PROGRAM EM02_Placing1
VAR
	
	//Backbone
	FB_StateMachine_Placing1		: FB_StateManager;
	bFl_RunningMachinePlacing1		: BOOL;
	bFl_SeqReset					: BOOL;
	bFl_Manual						: BOOL;
	CheckStatusPlacing1				: checkstatus;
	AlarmEventHistory				: ARRAY[1..20] OF Alarm_Event_History;
	Placing1_Management				: FB_Placing_v2;
	bFl_Flushing					: BOOL;
	PalletID_Placing1				: PalletID_name;
	Placing1_ID						: STRING;
	bFl_PalletJammed				: BOOL;
	
	//Motor
	Motor_PalletPlacing1			: MotorManagement;
	bFl_MotorPlacing1				: BOOL;
	Motor_Placing1_Error			: BOOL;
	Motor_Placing1_ErrorID			: UINT;
	bFl_MotorPlacing1_Fwd			: BOOL;
	bFl_MotorPlacing1_Rev			: BOOL;
	bFL_Safety						: BOOL;
	AlarmEventActive				: ARRAY[1..20] OF Alarm_Event_Active;
	CheckAcc						: TON;
END_VAR
VAR // added by the converter: edge detectors and wires of the graphical bodies
    _w1 : BOOL;
END_VAR

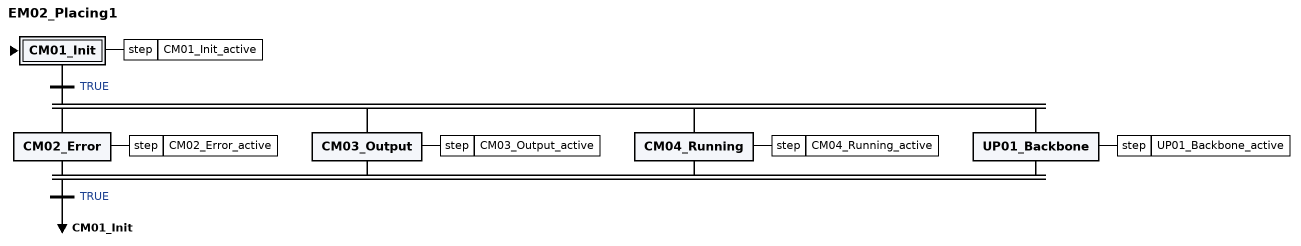
INITIAL_STEP CM01_Init:
    CM01_Init_active(N);  // step action
END_STEP
TRANSITION FROM CM01_Init TO (CM02_Error, CM03_Output, CM04_Running, UP01_Backbone)
    := TRUE;
END_TRANSITION
STEP CM02_Error:
    CM02_Error_active(N);  // step action
END_STEP
STEP CM03_Output:
    CM03_Output_active(N);  // step action
END_STEP
STEP CM04_Running:
    CM04_Running_active(N);  // step action
END_STEP
STEP UP01_Backbone:
    UP01_Backbone_active(N);  // step action
END_STEP
TRANSITION FROM (CM02_Error, CM03_Output, CM04_Running, UP01_Backbone) TO CM01_Init
    := TRUE;
END_TRANSITION

ACTION CM01_Init_active:
Data_GVL.bFL_StartPlacing1			:= Status_GVL.bFl_RunButton_Robotic OR HMI_GVL.bStartButtonPlacing1;
Data_GVL.bFL_StopPlacing1			:= NOT Status_GVL.bFl_StopButton_Robotic OR HMI_GVL.bStopButtonPlacing1;
Data_GVL.bFL_ResetPlacing1			:= Status_GVL.bFl_ResetButton_Robotic OR HMI_GVL.bResetButtonPlacing1;
Data_GVL.bFL_AckPlacing1			:= Status_GVL.bFl_Acknowledge_Robotic OR HMI_GVL.bAcknowledgeButtonPlacing1;
Data_GVL.bFL_AutoManuaModePlacing1 	:= Status_GVL.bFl_Manual_Robotic OR HMI_GVL.bTestModeEnablePlacing1;
bFl_RunningMachinePlacing1			:= Data_GVL.stStateMachinePlacing1.Running;
bFl_Manual							:= Data_GVL.stStateMachinePlacing1.ManualMode;
bFl_SeqReset						:= NOT Status_GVL.bFl_EStop_Robotic;
bFL_Safety							:= Status_GVL.bFl_EStop_Robotic AND Status_GVL.bSafety_DoorRobotic;


(*=================Convert Timer============================*)
Data_GVL.Tmr_Placing1	:= ConvertMilliSecTimeData(HMI_GVL.Tmr_Placing1);

(*=================Data OEE============================*)
Data_GVL.dt_Production[1].Data1			:= HMI_GVL.arCountTotal[1];
Data_GVL.dt_Production[1].Data2			:= HMI_GVL.arPalletTotal[1];
Data_GVL.dt_Production[1].Data3			:= HMI_GVL.arPalletIncomplete[1];
Data_GVL.dt_Production[1].ProductCode	:= Status_GVL.RecipeLine[1].ProductName;
END_ACTION

ACTION CM02_Error_active:
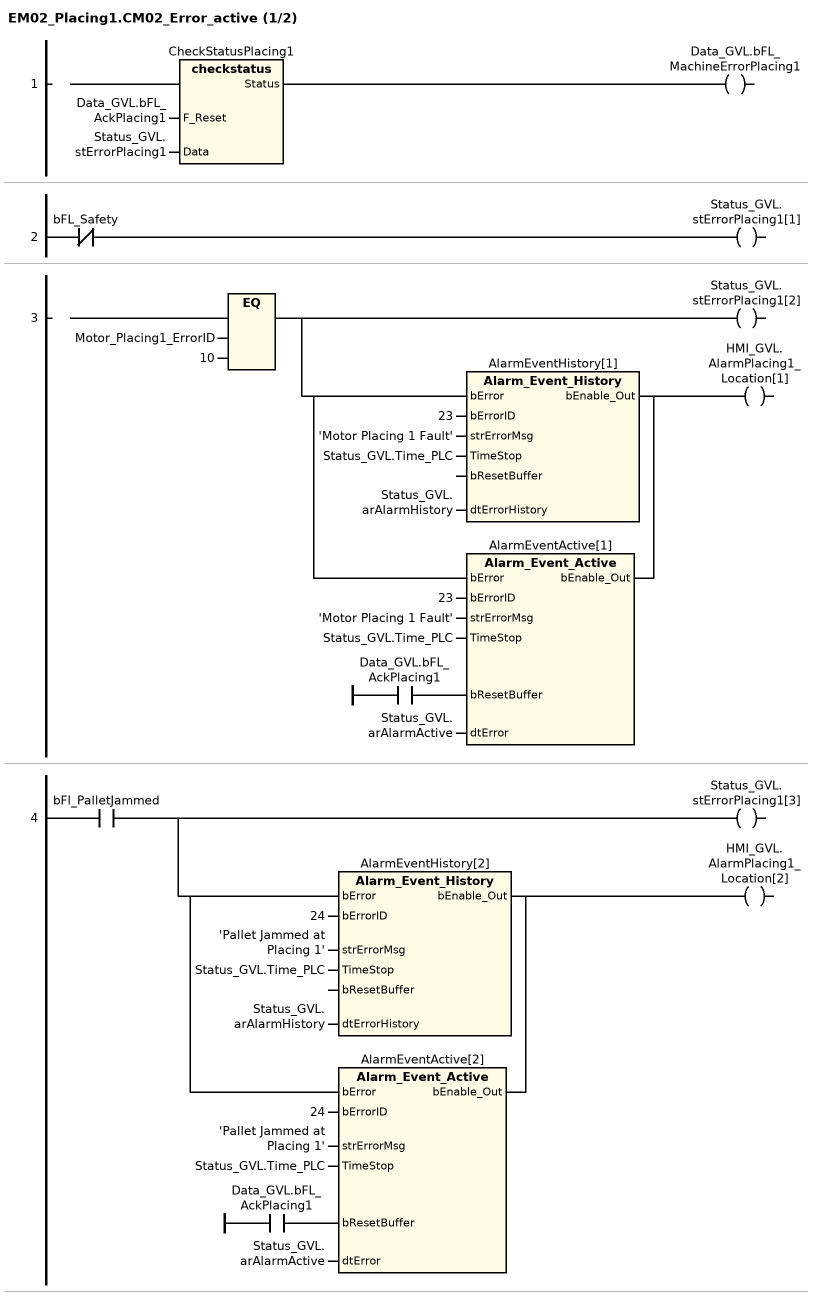
// NETWORK 1
CheckStatusPlacing1(F_Reset := Data_GVL.bFL_AckPlacing1, Data := Status_GVL.stErrorPlacing1); // checkstatus
Data_GVL.bFL_MachineErrorPlacing1 := CheckStatusPlacing1.Status;

// NETWORK 2
Status_GVL.stErrorPlacing1[1] := NOT bFL_Safety;

// NETWORK 3
_w1 := Motor_Placing1_ErrorID = 10;
Status_GVL.stErrorPlacing1[2] := _w1;
AlarmEventHistory[1](
    bError := _w1,
    bErrorID := 23,
    strErrorMsg := 'Motor Placing 1 Fault',
    TimeStop := Status_GVL.Time_PLC,
    dtErrorHistory := Status_GVL.arAlarmHistory); // Alarm_Event_History
AlarmEventActive[1](
    bError := _w1,
    bErrorID := 23,
    strErrorMsg := 'Motor Placing 1 Fault',
    TimeStop := Status_GVL.Time_PLC,
    bResetBuffer := Data_GVL.bFL_AckPlacing1,
    dtError := Status_GVL.arAlarmActive); // Alarm_Event_Active
HMI_GVL.AlarmPlacing1_Location[1] := AlarmEventHistory[1].bEnable_Out OR AlarmEventActive[1].bEnable_Out;

// NETWORK 4
Status_GVL.stErrorPlacing1[3] := bFl_PalletJammed;
AlarmEventHistory[2](
    bError := bFl_PalletJammed,
    bErrorID := 24,
    strErrorMsg := 'Pallet Jammed at Placing 1',
    TimeStop := Status_GVL.Time_PLC,
    dtErrorHistory := Status_GVL.arAlarmHistory); // Alarm_Event_History
AlarmEventActive[2](
    bError := bFl_PalletJammed,
    bErrorID := 24,
    strErrorMsg := 'Pallet Jammed at Placing 1',
    TimeStop := Status_GVL.Time_PLC,
    bResetBuffer := Data_GVL.bFL_AckPlacing1,
    dtError := Status_GVL.arAlarmActive); // Alarm_Event_Active
HMI_GVL.AlarmPlacing1_Location[2] := AlarmEventHistory[2].bEnable_Out OR AlarmEventActive[2].bEnable_Out;

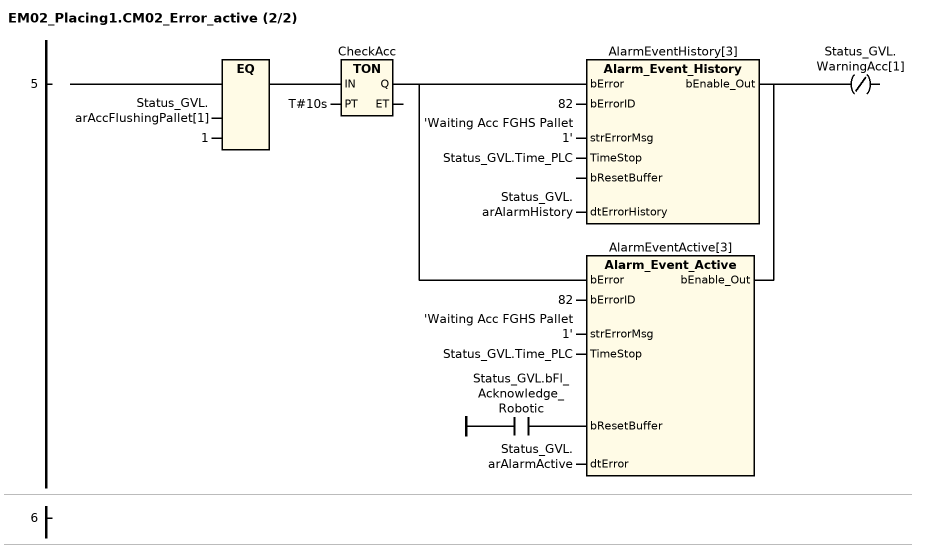
// NETWORK 5
CheckAcc(IN := Status_GVL.arAccFlushingPallet[1] = 1, PT := T#10s); // TON
AlarmEventHistory[3](
    bError := CheckAcc.Q,
    bErrorID := 82,
    strErrorMsg := 'Waiting Acc FGHS Pallet 1',
    TimeStop := Status_GVL.Time_PLC,
    dtErrorHistory := Status_GVL.arAlarmHistory); // Alarm_Event_History
AlarmEventActive[3](
    bError := CheckAcc.Q,
    bErrorID := 82,
    strErrorMsg := 'Waiting Acc FGHS Pallet 1',
    TimeStop := Status_GVL.Time_PLC,
    bResetBuffer := Status_GVL.bFl_Acknowledge_Robotic,
    dtError := Status_GVL.arAlarmActive); // Alarm_Event_Active
Status_GVL.WarningAcc[1] := NOT (AlarmEventHistory[3].bEnable_Out OR AlarmEventActive[3].bEnable_Out);

// NETWORK 6
END_ACTION

ACTION CM03_Output_active:
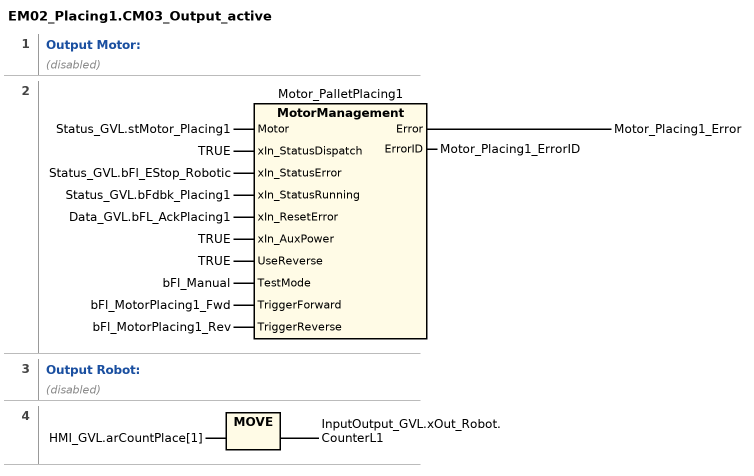
// NETWORK 1 (disabled)
// label: Output Motor

// NETWORK 2
Motor_PalletPlacing1(
    Motor := Status_GVL.stMotor_Placing1,
    xIn_StatusDispatch := TRUE,
    xIn_StatusError := Status_GVL.bFl_EStop_Robotic,
    xIn_StatusRunning := Status_GVL.bFdbk_Placing1,
    xIn_ResetError := Data_GVL.bFL_AckPlacing1,
    xIn_AuxPower := TRUE,
    UseReverse := TRUE,
    TestMode := bFl_Manual,
    TriggerForward := bFl_MotorPlacing1_Fwd,
    TriggerReverse := bFl_MotorPlacing1_Rev,
    ErrorID => Motor_Placing1_ErrorID); // MotorManagement
Motor_Placing1_Error := Motor_PalletPlacing1.Error;

// NETWORK 3 (disabled)
// label: Output Robot

// NETWORK 4
InputOutput_GVL.xOut_Robot.CounterL1 := HMI_GVL.arCountPlace[1];
END_ACTION

ACTION CM04_Running_active:
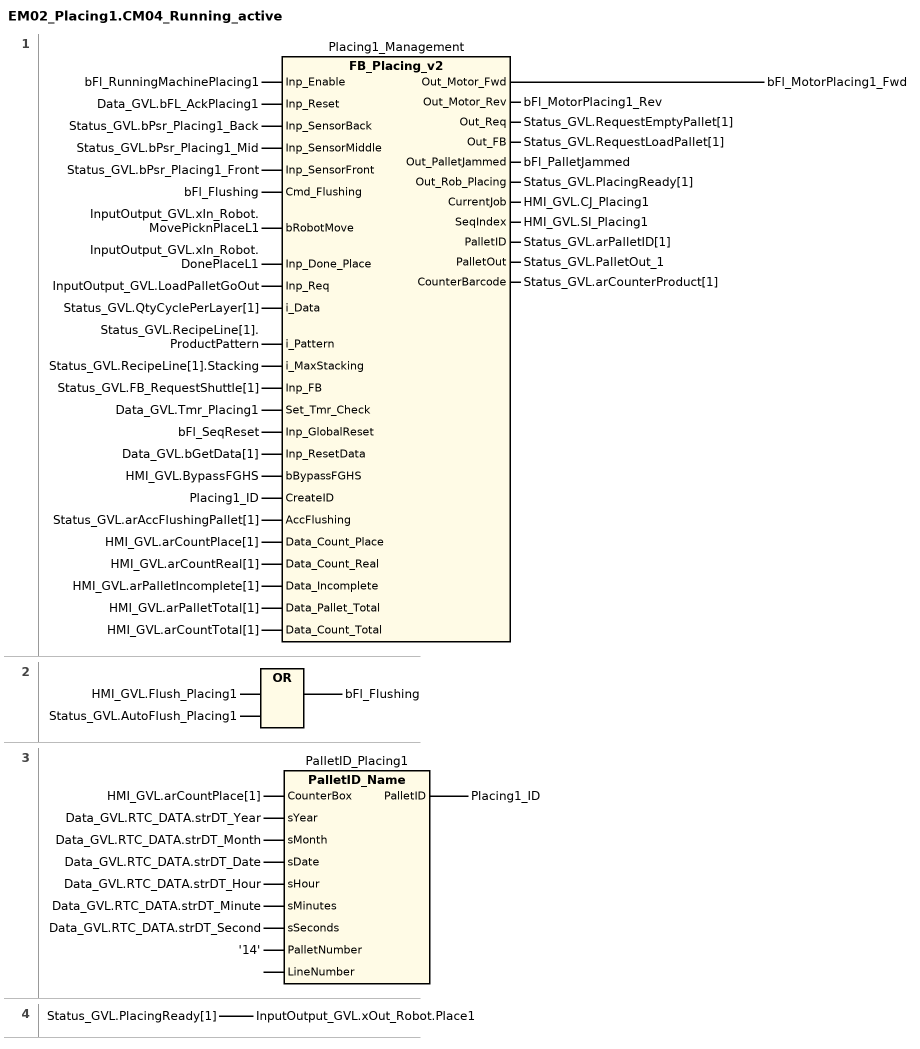
// NETWORK 1
Placing1_Management(
    Inp_Enable := bFl_RunningMachinePlacing1,
    Inp_Reset := Data_GVL.bFL_AckPlacing1,
    Inp_SensorBack := Status_GVL.bPsr_Placing1_Back,
    Inp_SensorMiddle := Status_GVL.bPsr_Placing1_Mid,
    Inp_SensorFront := Status_GVL.bPsr_Placing1_Front,
    Cmd_Flushing := bFl_Flushing,
    bRobotMove := InputOutput_GVL.xIn_Robot.MovePicknPlaceL1,
    Inp_Done_Place := InputOutput_GVL.xIn_Robot.DonePlaceL1,
    Inp_Req := InputOutput_GVL.LoadPalletGoOut,
    i_Data := Status_GVL.QtyCyclePerLayer[1],
    i_Pattern := Status_GVL.RecipeLine[1].ProductPattern,
    i_MaxStacking := Status_GVL.RecipeLine[1].Stacking,
    Inp_FB := Status_GVL.FB_RequestShuttle[1],
    Set_Tmr_Check := Data_GVL.Tmr_Placing1,
    Inp_GlobalReset := bFl_SeqReset,
    Inp_ResetData := Data_GVL.bGetData[1],
    bBypassFGHS := HMI_GVL.BypassFGHS,
    CreateID := Placing1_ID,
    AccFlushing := Status_GVL.arAccFlushingPallet[1],
    Data_Count_Place := HMI_GVL.arCountPlace[1],
    Data_Count_Real := HMI_GVL.arCountReal[1],
    Data_Incomplete := HMI_GVL.arPalletIncomplete[1],
    Data_Pallet_Total := HMI_GVL.arPalletTotal[1],
    Data_Count_Total := HMI_GVL.arCountTotal[1],
    Out_Motor_Rev => bFl_MotorPlacing1_Rev,
    Out_Req => Status_GVL.RequestEmptyPallet[1],
    Out_FB => Status_GVL.RequestLoadPallet[1],
    Out_PalletJammed => bFl_PalletJammed,
    Out_Rob_Placing => Status_GVL.PlacingReady[1],
    CurrentJob => HMI_GVL.CJ_Placing1,
    SeqIndex => HMI_GVL.SI_Placing1,
    PalletID => Status_GVL.arPalletID[1],
    PalletOut => Status_GVL.PalletOut_1,
    CounterBarcode => Status_GVL.arCounterProduct[1]); // FB_Placing_v2
bFl_MotorPlacing1_Fwd := Placing1_Management.Out_Motor_Fwd;

// NETWORK 2
bFl_Flushing := HMI_GVL.Flush_Placing1 OR Status_GVL.AutoFlush_Placing1;

// NETWORK 3
PalletID_Placing1(
    CounterBox := HMI_GVL.arCountPlace[1],
    sYear := Data_GVL.RTC_DATA.strDT_Year,
    sMonth := Data_GVL.RTC_DATA.strDT_Month,
    sDate := Data_GVL.RTC_DATA.strDT_Date,
    sHour := Data_GVL.RTC_DATA.strDT_Hour,
    sMinutes := Data_GVL.RTC_DATA.strDT_Minute,
    sSeconds := Data_GVL.RTC_DATA.strDT_Second,
    PalletNumber := '14'); // PalletID_Name
Placing1_ID := PalletID_Placing1.PalletID;

// NETWORK 4
InputOutput_GVL.xOut_Robot.Place1 := Status_GVL.PlacingReady[1];
END_ACTION

ACTION UP01_Backbone_active:
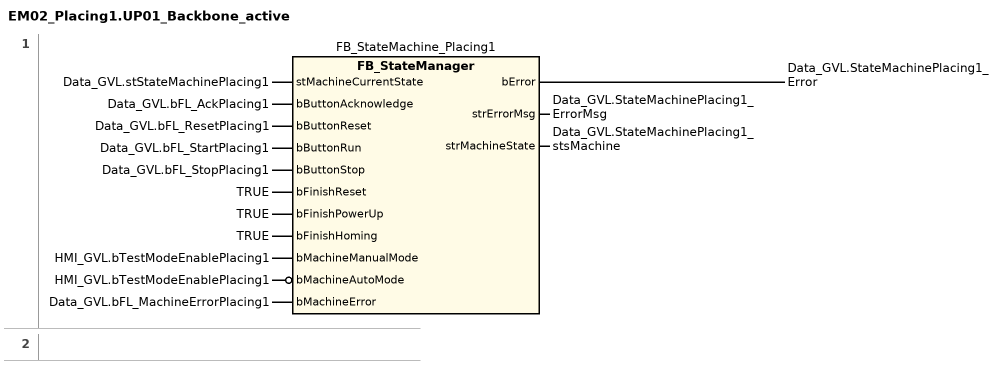
// NETWORK 1
FB_StateMachine_Placing1(
    stMachineCurrentState := Data_GVL.stStateMachinePlacing1,
    bButtonAcknowledge := Data_GVL.bFL_AckPlacing1,
    bButtonReset := Data_GVL.bFL_ResetPlacing1,
    bButtonRun := Data_GVL.bFL_StartPlacing1,
    bButtonStop := Data_GVL.bFL_StopPlacing1,
    bFinishReset := TRUE,
    bFinishPowerUp := TRUE,
    bFinishHoming := TRUE,
    bMachineManualMode := HMI_GVL.bTestModeEnablePlacing1,
    bMachineAutoMode := NOT HMI_GVL.bTestModeEnablePlacing1,
    bMachineError := Data_GVL.bFL_MachineErrorPlacing1,
    strErrorMsg => Data_GVL.StateMachinePlacing1_ErrorMsg,
    strMachineState => Data_GVL.StateMachinePlacing1_stsMachine); // FB_StateManager
Data_GVL.StateMachinePlacing1_Error := FB_StateMachine_Placing1.bError;

// NETWORK 2
END_ACTION

END_PROGRAM

(* stored: Version 1.1.0.1, ProductVersion 3.1.4024.12
   POU EM02_Placing1: Id {00aa432e-e792-4c25-afb1-75848a64f778}, SpecialFunc None
   Action CM01_Init_active: Id {fc494458-a53a-47d4-9015-e1f63be3b838}
   Action CM02_Error_active: Id {5fa71375-e7f6-4084-ad7e-0e3dc8c2af73}
   Action CM03_Output_active: Id {72afaa0d-a9c7-4084-aa79-deb89f78f292}
   Action CM04_Running_active: Id {2e0bb76c-fe50-4766-aca4-71aa08bb3f3d}
   Action UP01_Backbone_active: Id {081eb043-5e45-4398-9983-10616fdc2eca} *)
